// TIA Portal V15.1 export
// export: Created 2024-06-21T08:40:40.7968835Z, ExportSetting WithDefaults, DisplayName Totally Integrated Automation Portal, DisplayVersion V15.1 Update 5, DisplayName TIA Portal Openness, DisplayVersion V15.1 Update 5, DisplayName SINAMICS Startdrive Advanced, DisplayVersion V15.1, DisplayName G130, G150, S120, S150, SINAMICS MV, S210, DisplayVersion V15.1, DisplayName G110M, G120, G120C, G120D, G120P, DisplayVersion V15.1, DisplayName STEP 7 Professional, DisplayVersion V15.1 Update 5, DisplayName STEP 7 Safety, DisplayVersion V15.1, DisplayName WinCC Professional, DisplayVersion V15.1 Update 5, DisplayName SIMATIC Visualization Architect, DisplayVersion V15.1
DATA_BLOCK "_209000NCP01AE"   // DB253
{ S7_Optimized_Access := 'FALSE' }
AUTHOR : VCC
NAME : LocFnc
VERSION : 0.1
// stored: AutoNumber false, DBAccessibleFromOPCUA true, IsOnlyStoredInLoadMemory false, IsWriteProtectedInAS false
   VAR RETAIN
      AA_AE01E1QM1 { ExternalAccessible := 'False'; ExternalVisible := 'False'; ExternalWritable := 'False'} : Bool;   // AE01 EG1 - Overload protection power supply 24VDC
      AA_AE01E3EG1 { ExternalAccessible := 'False'; ExternalVisible := 'False'; ExternalWritable := 'False'} : Bool;   // AE01 EG1 - Power supply 24VDC NOK
      AD_AE01E3FV1 { ExternalAccessible := 'False'; ExternalVisible := 'False'; ExternalWritable := 'False'} : Bool;   // AE01 EG1 - Surge protection 24VDC NOK
      AC_AE01E3FS31 { ExternalAccessible := 'False'; ExternalVisible := 'False'; ExternalWritable := 'False'} : Bool;   // 24VDC Fuse - Gateway 24VDC electronic fuses AE01-JC31
      AA_AE01E3FS01_CH1 { ExternalAccessible := 'False'; ExternalVisible := 'False'; ExternalWritable := 'False'} : Bool;   // 24VDC Fuse - General - PLC
      AC_AE01E3FS01_CH2 { ExternalAccessible := 'False'; ExternalVisible := 'False'; ExternalWritable := 'False'} : Bool;   // 24VDC Fuse - General - Measuring point PNMA II
      AA_AE01E3FS02_CH1 { ExternalAccessible := 'False'; ExternalVisible := 'False'; ExternalWritable := 'False'} : Bool;   // 24VDC Fuse - General - Scalance 1
      AA_AE01E3FS02_CH2 { ExternalAccessible := 'False'; ExternalVisible := 'False'; ExternalWritable := 'False'} : Bool;   // 24VDC Fuse - General - Scalance 2
      AA_AE01E3FS03_CH1 { ExternalAccessible := 'False'; ExternalVisible := 'False'; ExternalWritable := 'False'} : Bool;   // 24VDC Fuse - General - PN/PN Couplers AE02
      AA_AE01E3FS03_CH2 { ExternalAccessible := 'False'; ExternalVisible := 'False'; ExternalWritable := 'False'} : Bool;   // 24VDC Fuse - General - Busnode + Com. PLC212
      AC_AE01E3FS04_CH1 { ExternalAccessible := 'False'; ExternalVisible := 'False'; ExternalWritable := 'False'} : Bool;   // 24VDC Fuse - General - ETA Gateway AK02
      AA_AE01E3FS04_CH2 { ExternalAccessible := 'False'; ExternalVisible := 'False'; ExternalWritable := 'False'} : Bool;   // 24VDC Fuse - General - Busnodes AK
      AA_AE01E3FS05_CH1 { ExternalAccessible := 'False'; ExternalVisible := 'False'; ExternalWritable := 'False'} : Bool;   // 24VDC Fuse - General - Busnode General Field
      AD_AE01E3FS01_CH1 { ExternalAccessible := 'False'; ExternalVisible := 'False'; ExternalWritable := 'False'} : Bool;   // 24VDC Fuse - General - PLC
      AD_AE01E3FS01_CH2 { ExternalAccessible := 'False'; ExternalVisible := 'False'; ExternalWritable := 'False'} : Bool;   // 24VDC Fuse - General - Measuring point PNMA II
      AD_AE01E3FS02_CH1 { ExternalAccessible := 'False'; ExternalVisible := 'False'; ExternalWritable := 'False'} : Bool;   // 24VDC Fuse - General - Scalance 1
      AD_AE01E3FS02_CH2 { ExternalAccessible := 'False'; ExternalVisible := 'False'; ExternalWritable := 'False'} : Bool;   // 24VDC Fuse - General - Scalance 2
      AD_AE01E3FS03_CH1 { ExternalAccessible := 'False'; ExternalVisible := 'False'; ExternalWritable := 'False'} : Bool;   // 24VDC Fuse - General - PN/PN Couplers AE02
      AD_AE01E3FS03_CH2 { ExternalAccessible := 'False'; ExternalVisible := 'False'; ExternalWritable := 'False'} : Bool;   // 24VDC Fuse - General - Busnode + Com. PLC212
      AD_AE01E3FS04_CH1 { ExternalAccessible := 'False'; ExternalVisible := 'False'; ExternalWritable := 'False'} : Bool;   // 24VDC Fuse - General - ETA Gateway AK02
      AD_AE01E3FS04_CH2 { ExternalAccessible := 'False'; ExternalVisible := 'False'; ExternalWritable := 'False'} : Bool;   // 24VDC Fuse - General - Busnodes AK
      AD_AE01E3FS05_CH1 { ExternalAccessible := 'False'; ExternalVisible := 'False'; ExternalWritable := 'False'} : Bool;   // 24VDC Fuse - General - Busnode General Field
      AC_AE01EL1 { ExternalAccessible := 'False'; ExternalVisible := 'False'; ExternalWritable := 'False'} : Bool;   // Fault heat exchanger cabinet AE01
      AD_AE01E2SG1 { ExternalAccessible := 'False'; ExternalVisible := 'False'; ExternalWritable := 'False'} : Bool;   // Door not closed cabinet AE01
      AD_AE02E2SG1 { ExternalAccessible := 'False'; ExternalVisible := 'False'; ExternalWritable := 'False'} : Bool;   // Door not closed cabinet AE02
      AC_AE01QC1 { ExternalAccessible := 'False'; ExternalVisible := 'False'; ExternalWritable := 'False'} : Bool;   // Contactor summary door closed not ok, cabinet AE01-AE02
      AE01E1QM1AlarmABCondition { ExternalAccessible := 'False'; ExternalVisible := 'False'; ExternalWritable := 'False'} : Bool;   // Alarm AB condition
      AE01E3EG1AlarmABCondition { ExternalAccessible := 'False'; ExternalVisible := 'False'; ExternalWritable := 'False'} : Bool;   // Alarm AB condition
      AE01E3FS01_CH1AlarmABCondition { ExternalAccessible := 'False'; ExternalVisible := 'False'; ExternalWritable := 'False'} : Bool;   // Alarm AB condition
      AE01E3FS02_CH1AlarmABCondition { ExternalAccessible := 'False'; ExternalVisible := 'False'; ExternalWritable := 'False'} : Bool;   // Alarm AB condition
      AE01E3FS02_CH2AlarmABCondition { ExternalAccessible := 'False'; ExternalVisible := 'False'; ExternalWritable := 'False'} : Bool;   // Alarm AB condition
      AE01E3FS03_CH1AlarmABCondition { ExternalAccessible := 'False'; ExternalVisible := 'False'; ExternalWritable := 'False'} : Bool;   // Alarm AB condition
      AE01E3FS03_CH2AlarmABCondition { ExternalAccessible := 'False'; ExternalVisible := 'False'; ExternalWritable := 'False'} : Bool;   // Alarm AB condition
      AE01E3FS04_CH2AlarmABCondition { ExternalAccessible := 'False'; ExternalVisible := 'False'; ExternalWritable := 'False'} : Bool;   // Alarm AB condition
      AE01E3FS05_CH1AlarmABCondition { ExternalAccessible := 'False'; ExternalVisible := 'False'; ExternalWritable := 'False'} : Bool;   // Alarm AB condition
      H_209000AE01E1QM1IAnim : Word;   // HMI Animation of the icon
      H_209000AE01E3EG1IAnim : Word;   // HMI Animation of the icon
      H_209000AE01E3FV1IAnim : Word;   // HMI Animation of the icon
      H_209000AE01E3CE1IAnim : Word;   // HMI Animation of the icon
      H_209000AE01E3FS31IAnim : Word;   // HMI Animation of the icon
      H_209000AE01E3FS01_CH1IAnim : Word;   // HMI Animation of the icon
      H_209000AE01E3FS01_CH2IAnim : Word;   // HMI Animation of the icon
      H_209000AE01E3FS02_CH1IAnim : Word;   // HMI Animation of the icon
      H_209000AE01E3FS02_CH2IAnim : Word;   // HMI Animation of the icon
      H_209000AE01E3FS03_CH1IAnim : Word;   // HMI Animation of the icon
      H_209000AE01E3FS03_CH2IAnim : Word;   // HMI Animation of the icon
      H_209000AE01E3FS04_CH1IAnim : Word;   // HMI Animation of the icon
      H_209000AE01E3FS04_CH2IAnim : Word;   // HMI Animation of the icon
      H_209000AE01E3FS05_CH1IAnim : Word;   // HMI Animation of the icon
      H_209000AE01E3FS05_CH2IAnim : Word;   // HMI Animation of the icon
      H_209000AE01EL1IAnim : Word;   // HMI Animation of the icon
      H_209000AE01E2SG1IAnim : Word;   // HMI Animation of the icon
      H_209000AE02E2SG1IAnim : Word;   // HMI Animation of the icon
      H_209000AE01QC1IAnim : Word;   // HMI Animation of the icon
      H_DBnr : Int;   // DB number
      H_Anim : Word;   // Animation
      H_HMI : Struct   // Icon Animation
         "209000AE01JC31" : "H_HMI";   // HMI Animation of the icon
      END_STRUCT;
      H : Struct   // Animation
         "209000AE01JC31" : "H_ETAFuseCPC20PN";   // HMI Animation
      END_STRUCT;
      AlarmA { ExternalAccessible := 'False'; ExternalVisible := 'False'; ExternalWritable := 'False'} : Bool;   // Alarm A
      AlarmB { ExternalAccessible := 'False'; ExternalVisible := 'False'; ExternalWritable := 'False'} : Bool;   // Alarm B
      AlarmC { ExternalAccessible := 'False'; ExternalVisible := 'False'; ExternalWritable := 'False'} : Bool;   // Alarm C
      AlarmD { ExternalAccessible := 'False'; ExternalVisible := 'False'; ExternalWritable := 'False'} : Bool;   // Alarm D
      AlarmABCondition { ExternalAccessible := 'False'; ExternalVisible := 'False'; ExternalWritable := 'False'} : Bool;   // Alarm AB condition
      AE01E3CE1Active { ExternalAccessible := 'False'; ExternalVisible := 'False'; ExternalWritable := 'False'} : Bool;   // Buffer Module active
      AE01E3CE1 { ExternalAccessible := 'False'; ExternalVisible := 'False'; ExternalWritable := 'False'} : "AlarmBits";   // Buffer module Alarm Bits
      "AE01-JC31" { ExternalAccessible := 'False'; ExternalVisible := 'False'; ExternalWritable := 'False'} : "AlarmBits";   // ETA fuse Alarm Bits
      "AE01-JC31_ETAFuseData" { ExternalAccessible := 'False'; ExternalVisible := 'False'; ExternalWritable := 'False'} : "ETAFuseData";   // ETA fuse status
   END_VAR
BEGIN
END_DATA_BLOCK
